FUNCTION INTERNAL _Cleanup
VAR
	i					: UDINT;
	_iSignal			: I_SignalNode;
END_VAR

// Loop through stEntry to update signal ids
FOR i := 1 TO Param.BROADCAST_CAP DO
	IF _Broadcast.stEntry[i].iSignal <> 0 AND_THEN _Broadcast.stEntry[i].iSignal <> _iSignal THEN
			_iSignal := _Broadcast.stEntry[i].iSignal;
			_iSignal.id := i;
	END_IF
END_FOR

END_FUNCTION

(* stored: Version 1.1.0.1
   POU _Cleanup: Id {a89a05f8-a071-481e-a16c-f3ed21348be6}, SpecialFunc None *)
